SYSTEM TEST_VSTYLE (* Test Display of VSTYLE values *)
  (* Standard: 61499-1 *)
  (* Version 0.0, 2000-05-27, JHC, Rockwell Automation *)
  DEVICE HMI : FRAME_DEVICE(BOUNDS := [100,100,330,80])
    RESOURCE RES1 : PANEL_RESOURCE
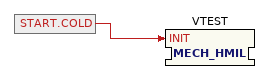
      FBS
        VTEST : MECH_HMIL;
      END_FBS
      EVENT_CONNECTIONS
        START.COLD TO VTEST.INIT;
      END_CONNECTIONS
    END_RESOURCE
  END_DEVICE
  DEVICE VIEW : FRAME_DEVICE(BOUNDS := [430,100,40,175])
    RESOURCE RES1 : PANEL_RESOURCE
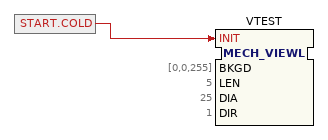
      FBS
        VTEST : MECH_VIEWL(BKGD := [0,0,255], LEN := 5, DIA := 25, DIR := 1);
      END_FBS
      EVENT_CONNECTIONS
        START.COLD TO VTEST.INIT;
      END_CONNECTIONS
    END_RESOURCE
  END_DEVICE
END_SYSTEM
